TYPE ST_CSV_Record :
STRUCT
	sName 	: T_MaxString 	:= '';
	nNumber	: UDINT 		:= 0;
	fPos		: LREAL 		:= 0.0;
	bOP		: BOOL 		:= FALSE;
	sDesc		: STRING(40)	:= '';
	data		: ARRAY[0..7] OF BYTE;
END_STRUCT
END_TYPE

(* stored: Version 1.1.0.1, ProductVersion 3.1.4024.9
   DUT ST_CSV_Record: Id {540041e3-1efc-4949-a732-2d231ae8b0ea} *)
